TYPE csp_case_loader_status_enum :
(
	CSP_CASE_LOADER_STATUS_NOT_INITIALIZED 							:=  0,
	CSP_CASE_LOADER_STATUS_DISABLED 								:=  10,
	CSP_CASE_LOADER_STATUS_ENABLE_REQUEST 							:=  20,
	CSP_CASE_LOADER_STATUS_ENABLING 								:=  30,
	CSP_CASE_LOADER_STATUS_ENABLED 									:=  40,
	CSP_CASE_LOADER_STATUS_CHANGE_OVER_MODE							:=  45,
	CSP_CASE_LOADER_STATUS_ENABLE_CROSSPUSHERS						:=  46,
	CSP_CASE_LOADER_STATUS_MOVE_CROSSPUSHERS						:=  47,
	CSP_CASE_LOADER_STATUS_VERIFY_CROSSPUSHERS_CLEAR				:=  48,
	CSP_CASE_LOADER_STATUS_MOVE_AXIS_TO_POS							:=  49,
	CSP_CASE_LOADER_STATUS_HOME_REQUEST								:=  50,
	CSP_CASE_LOADER_STATUS_HOMING									:=  60,
	CSP_CASE_LOADER_STATUS_HOME_DONE								:=  70,
	CSP_CASE_LOADER_STATUS_LENGTH_MOVE_TO_CLEAR_POS					:=  80,
	CSP_CASE_LOADER_STATUS_LENGTH_MOVING_TO_CLEAR_POS				:=  85,
	CSP_CASE_LOADER_STATUS_LENGTH_WAITING_FOR_GUIDES_TO_PHASE		:=  87,
	CSP_CASE_LOADER_STATUS_CALCULATING_SLAVE_POSITION				:=  90,
	CSP_CASE_LOADER_STATUS_CALCULATING_MASTER_POSITION				:=  91,
	CSP_CASE_LOADER_STATUS_WAITING_SLAVE_ENGAGE						:= 100,
	CSP_CASE_LOADER_STATUS_WAITING_MASTER_ENGAGE					:= 101,
	CSP_CASE_LOADER_STATUS_LOADER_PLATE_PHASE_REQUIRED				:= 130,
	CSP_CASE_LOADER_STATUS_PHASE_REQUEST							:= 140,
	CSP_CASE_LOADER_STATUS_PHASING									:= 150,
	CSP_CASE_LOADER_STATUS_PHASED									:= 160,
	CSP_CASE_LOADER_STATUS_CAM_ENGAGED_REQ							:= 170,
	CSP_CASE_LOADER_STATUS_AXIS_ENGAGE_VERIFY						:= 180,
	CSP_CASE_LOADER_STATUS_CAM_ENGAGED								:= 190,
	CSP_CASE_LOADER_STATUS_CAM_TABLE_READ							:= 195,
	CSP_CASE_LOADER_STATUS_CALCULATE_SLAVE_POSITION_REQUEST			:= 196,
	CSP_CASE_LOADER_STATUS_READY									:= 197,
	CSP_CASE_LOADER_STATUS_RUNNING									:= 200,
	CSP_CASE_LOADER_STATUS_MOVING									:= 205,
	CSP_CASE_LOADER_STATUS_DISENGAGE_REQUEST						:= 210,
	CSP_CASE_LOADER_STATUS_DISENGAGING								:= 211,	
	CSP_CASE_LOADER_STATUS_STOP_REQUEST 							:= 500,
	CSP_CASE_LOADER_STATUS_DISABLE_REQUEST 							:= 530,
	CSP_CASE_LOADER_STATUS_DISABLING 								:= 540,
	
	CSP_CASE_LOADER_STATUS_IMMEDIATE_DWELL_FOR_CASE_ALREADY_LOADED	:= 560,
	CSP_CASE_LOADER_STATUS_WAIT_FOR_REJECT_DONE						:= 565,
	CSP_CASE_LOADER_STATUS_WAIT_FOR_STACK_AT_LOADER					:= 570,
	CSP_CASE_LOADER_STATUS_FINISH_LOAD_CYCLE						:= 575,
	CSP_CASE_LOADER_STATUS_WAIT_FOR_NEW_LOAD						:= 580,
	CSP_CASE_LOADER_STATUS_LOAD_COMPLETE							:= 585,
	
	CSP_CASE_LOADER_STATUS_IMMEDIATE_DWELL_FOR_REJECT				:= 600,
	CSP_CASE_LOADER_STATUS_WAIT_FOR_REJECT_COMPLETE					:= 610,
	CSP_CASE_LOADER_STATUS_WAIT_FOR_LOAD							:= 620,
	CSP_CASE_LOADER_STATUS_VERIFY_SLAVES_ENGAGED					:= 630,
	CSP_CASE_LOADER_STATUS_RUN_LOAD_CYCLE							:= 640,
	CSP_CASE_LOADER_STATUS_ENGAGE_TO_CASE_VM						:= 650,
	
	CSP_CASE_LOADER_STATUS_IMMEDIATE_DISENGAGE_THEN_WAIT_CAM		:= 700,
	CSP_CASE_LOADER_STATUS_IMMEDIATE_DISENGAGE_CHECK_ZERO			:= 701,
	CSP_CASE_LOADER_STATUS_IMMEDIATE_DISENGAGE_MOVE_TO_ZERO			:= 702,
	CSP_CASE_LOADER_STATUS_IMMEDIATE_DISENGAGE_WAIT_MOVE			:= 703
	
) := CSP_CASE_LOADER_STATUS_NOT_INITIALIZED;
END_TYPE

(* stored: Version 1.1.0.1, ProductVersion 3.1.4024.3
   DUT csp_case_loader_status_enum: Id {cb28efae-8a23-45ca-809a-4b170f0e30b6} *)
